{attribute 'qualified_only'}
{attribute 'strict'}
TYPE MC_Source :
(
	mcSetValue := 0,
	mcActualValue := 1
);
END_TYPE

(* stored: Version 1.1.0.1, ProductVersion 3.1.4024.12
   DUT MC_Source: Id {7bb4e7c4-8f46-4691-9676-2ed94044bc38} *)
